// TIA Portal V16 export
// export: Created 2021-09-07T10:36:59.2550932Z, ExportSetting WithDefaults, DisplayName Totally Integrated Automation Portal, DisplayVersion V16 Update 3, DisplayName TIA Portal Version Control Interface, DisplayVersion V16 Update 2, DisplayName TIA Portal Openness, DisplayVersion V16 Update 3, DisplayName TIA Portal Teamcenter Gateway, DisplayVersion V16, DisplayName STEP 7 Professional, DisplayVersion V16 Update 3, DisplayName STEP 7 Safety, DisplayVersion V16, DisplayName WinCC Advanced, DisplayVersion V16 Update 3
FUNCTION_BLOCK "VolumeCounter"   // FB65, FBD
{ S7_Optimized_Access := 'TRUE' }
VERSION : 0.1
// stored: AutoNumber true, IsIECCheckEnabled false, IsRetainMemResEnabled false, MemoryReserve 100, SetENOAutomatically false, UDAEnableTagReadback false
   VAR_INPUT
      puls : Bool;
      nextHour : Bool;
      nextDay : Bool;
   END_VAR
   VAR_IN_OUT
      data : "FREQ_COUNTER";
   END_VAR
   VAR
      litrs : UInt;
      pTrig : Bool;
   END_VAR
   VAR CONSTANT
      FB_CALL_TIME : Real := 0.1;
   END_VAR
   VAR_TEMP   // added for the SCL form of the ladder/FBD networks
      _w1 : Bool;
   END_VAR
BEGIN

REGION Network 1: Add to counter
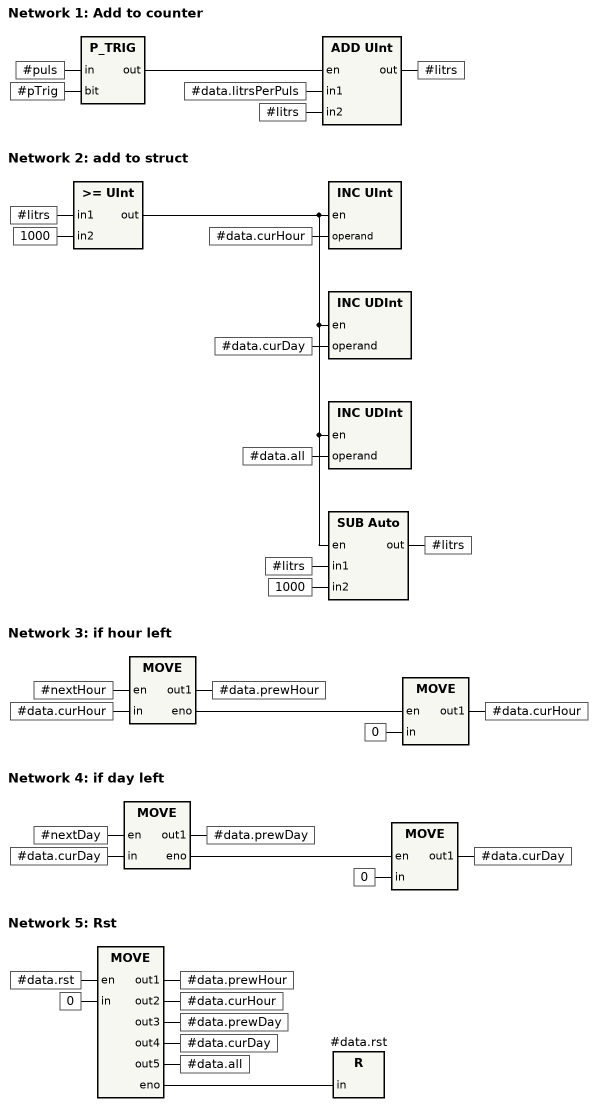
   #_w1 := #puls AND NOT #pTrig;   // rising edge
   #pTrig := #puls;
   IF #_w1 THEN #litrs := #data.litrsPerPuls + #litrs; END_IF;
END_REGION

REGION Network 2: add to struct
   IF #litrs >= 1000 THEN
       #data.curHour := #data.curHour + 1;
       #data.curDay := #data.curDay + 1;
       #data.all := #data.all + 1;
       #litrs := #litrs - 1000;
   END_IF;
END_REGION

REGION Network 3: if hour left
   IF #nextHour THEN
       #data.prewHour := #data.curHour;
       #data.curHour := 0;
   END_IF;
END_REGION

REGION Network 4: if day left
   IF #nextDay THEN
       #data.prewDay := #data.curDay;
       #data.curDay := 0;
   END_IF;
END_REGION

REGION Network 5: Rst
   IF #data.rst THEN
       #data.prewHour := 0;
       #data.curHour := 0;
       #data.prewDay := 0;
       #data.curDay := 0;
       #data.all := 0;
       #data.rst := FALSE;
   END_IF;
END_REGION
END_FUNCTION_BLOCK
